// ---- POUs/_Grundfunktionen/FB_Heizregler.TcPOU
FUNCTION_BLOCK FB_Heizregler
VAR_INPUT
	diTempSoll	: DINT;
	diTempIst 	: DINT;
	iTimeOffs 	: INT; (* 0..99 *)
	iTimeGrp		: INT; (* Auswahl der Timer-Gruppe 0..9 *)
	iPMin 			: INT := 25;
	iPMax 			: INT := 100;
	iPHeizIn		: INT := 0;
	bNewData		: BOOL;
END_VAR
VAR_OUTPUT
	iPHeizOut : INT;
END_VAR
VAR
	bInitDone					 : BOOL;

	(* %I / %Q ********************)
	QbOutHeizSteller		AT %Q* : BOOL;
	bOutHeizSteller		: BOOL;

	dwPWMfast					: DWORD;

	iPWMTimer					: INT;
	iPHeiz						: INT;

	adiTempIst 				: ARRAY[0..2] OF DINT;
	diTempIstAend 		: DINT;

	diTempSollOld 		: DINT;
	diTempSollAend 		: DINT;

	diTempDiff 				: DINT;

	diResult_P				: DINT;
	diResult_I				: DINT;
	diResult_Dist			: DINT;
	diResult_Dsoll		: DINT;
	diResult					: DINT;
END_VAR

VAR PERSISTENT
	bManuell	: BOOL;
	iManPHeiz : INT;

	dikP			: DINT := 300; (* P-Regler, 1000 = 1.000 *)
	dikI			: DINT := 50; (* I-Regler, 1000 = 1.000 *)
	dikDist		: DINT := 5; (* D-Regler auf Istwert *)
	dikDsoll	: DINT := 5; (* D-Regler auf Sollwert => wirkt direkt auf I-Anteil *)

END_VAR

IF NOT bInitDone THEN
	M_Init();
END_IF

M_Ctrl();
M_PWM();
M_PWMfast();

ACTION M_Ctrl:
IF bNewData THEN
	diTempSollAend :=
			diTempSoll
		- diTempSollOld;
	diTempSollOld := diTempSoll;
	diTempIstAend :=
			diTempIst
		- adiTempIst[2];
	adiTempIst[2] := adiTempIst[1];
	adiTempIst[1] := adiTempIst[0];
	adiTempIst[0] := diTempIst;
END_IF

IF NOT bManuell
AND NOT (iPHeizIn > 0)
AND gbHeizGruppe[iTimeGrp]
THEN
	IF bNewData THEN
		diResult_Dist :=
				diTempIstAend
			* dikDist;

		diResult_Dsoll :=
				diTempSollAend
			* dikDsoll;

		diTempDiff :=
				diTempSoll
			- diTempIst
			+ diResult_Dist;

		diResult_P :=
				diTempDiff
			* dikP;

		diResult_I :=
				diTempDiff
			* dikI
			+ diResult_Dsoll
			+ diResult_I;
		IF (diResult_I
				> (100000 - diResult_P))
		THEN
			diResult_I :=
				(100000 - diResult_P);
		ELSIF (diResult_I < 0) THEN
			diResult_I := 0;
		END_IF

		diResult :=
				diResult_P
			+ diResult_I;
		iPHeiz := DINT_TO_INT(diResult / 1000);

	END_IF

ELSE
	diResult_I := iManPHeiz * 1000;
	iPHeiz := iManPHeiz;
END_IF
END_ACTION

ACTION M_PWMfast:
(* PWM im SPS-Zyklus *)
IF bOutHeizSteller THEN
	dwPWMfast := dwPWMfast + 1;
	IF (dwPWMfast > gdwPWMfast_88) THEN
		QbOutHeizSteller := TRUE;
						(*	 dwPWMfast.1
						OR dwPWMfast.2
						OR dwPWMfast.3;*)
	ELSIF (dwPWMfast > gdwPWMfast_75) THEN
		QbOutHeizSteller :=
							 dwPWMfast.1
						OR dwPWMfast.2;
	ELSE
		QbOutHeizSteller :=
							dwPWMfast.1;
	END_IF
	dwPWMfast := dwPWMfast AND 16#00FFFFFF;
ELSE
	QbOutHeizSteller := FALSE;
	dwPWMfast := INT_TO_DWORD(iTimeOffs / 10);
END_IF
END_ACTION

ACTION M_PWM:
(* PWM-Funktion *)
IF gbPWMTakt THEN
	IF bManuell THEN
		iPHeiz := iManPHeiz;
	ELSIF (iPHeizIn > 0) THEN
		iPHeiz := iPHeizIn;
	END_IF
	IF iPHeiz > iPMax THEN
		iPHeiz := iPMax;
	END_IF
	IF (giPWMTimer = iTimeOffs) THEN
		iPWMTimer := 0;
		IF (iPHeiz > 0) AND gbHeizGruppe[iTimeGrp] THEN
			bOutHeizSteller := TRUE;
		END_IF
	END_IF
	IF bOutHeizSteller THEN
		IF (iPWMTimer > (iPHeiz + iPMin)) THEN
			bOutHeizSteller := FALSE;
		END_IF
		iPWMTimer := iPWMTimer + 1;
	ELSE
		iPWMTimer := 0;
	END_IF
END_IF
iPHeizOut := iPHeiz;
END_ACTION

ACTION M_Init:
IF bNewData THEN
	diTempSollOld := diTempSoll;
	adiTempIst[2] := diTempIst;
	adiTempIst[1] := diTempIst;
	adiTempIst[0] := diTempIst;
	diResult_I := iManPHeiz * 1000;
	bInitDone := TRUE;
END_IF
END_ACTION

END_FUNCTION_BLOCK

// ---- POUs/_Grundfunktionen/FB_Heizregler_FBHR.TcPOU
(* Heizregler fuer Fussbodenheizung ueber Schaltventil und 
	Ruecklauftemperaturueberwachung (Schwallbetrie)
*)
FUNCTION_BLOCK FB_Heizregler_FBHR
VAR_INPUT
	INbEnable				: BOOL;
	INrTempSoll			: REAL;
	INrTempIst 			: REAL;
	INrTempVorlauf	: REAL; (* Temperatur, Heizung Vorlauf *)
	INrTempFBHR			: REAL; (* Temperatur, Fussbodenheizung Ruecklauf*)

	iTimeGrp				: INT; (* Auswahl der Timer-Gruppe 0..9 *)
	iPMin 					: INT := 25;
	iPMax 					: INT := 100;
	iPHeizIn				: INT := 0;
END_VAR
VAR_OUTPUT
	iPHeizOut : INT;
END_VAR
VAR
	bInitDone					 : BOOL;

	(* %I / %Q ********************)
	QbOutHeizSteller		AT %Q* : BOOL;
	bOutHeizSteller		: BOOL;


	tonCtrlCycle			: TON := (PT:=T#5S);
	bCtrlCycle				: BOOL;
	rPHeiz						: REAL;

	arTempIst 				: ARRAY[0..2] OF REAL;
	rTempIstAend 			: REAL;

	rTempSollOld 			: REAL;
	rTempSollAend 		: REAL;

	rTempDiff 				: REAL;

	rResult_P					: REAL;
	rResult_I					: REAL;
	rResult_Dist			: REAL;
	rResult_Dsoll			: REAL;
	rResult						: REAL;
	
	iOutputState			: INT; (* Status der Ausgangssteuerung *)
	iOutputCycleTime	: INT; (* Zeit [s] seit dem letzten Heizvorgang *)
	rOutputCycleTime	: REAL; (* Zeit [%] seit dem letzten Heizvorgang *)
	tonTimeCycle						: TON := (PT:= T#1S); (* Zeittakt *)
	tofWasserHeizung				: TOF := (PT:= T#3S); (* Mindest-Einschaltzeit *)
	tonVorlaufTemp					: TON := (PT:= T#5M); (* maximale Wartezeit auf Vorlauftemperatur *)
	tonVorlaufTempStop			: TON := (PT:= T#15M); (* Wartezeit, wenn Vorlauftemperatur zu gering war *)
	tonMinWartezeit					: TON := (PT:= T#3M); (* Mindest-Wartezeit nach einem Heizyklus bis zum naechsten Start *)

	rRueckTempStart		: REAL; (* Ruecklauftemperatur beim Start des akt. Heizzyklusses *)

END_VAR

VAR PERSISTENT
	bManuell					: BOOL;
	iManPHeiz 				: INT;
	iMaxCycleTime			: INT := 3600; (* maximale Heizzykluszeit [s] bei Heizleistung 1% *)

	rkP								: REAL := 300; (* P-Regler, 1000 = 1.000 *)
	rkI								: REAL := 50; (* I-Regler, 1000 = 1.000 *)
	rkDist						: REAL := 5; (* D-Regler auf Istwert *)
	rkDsoll						: REAL := 5; (* D-Regler auf Sollwert => wirkt direkt auf I-Anteil *)

	rVorlTempDiffMin	: REAL := 5.0; (* Mindestdifferenz zwischen Vorlauf- und Raumtemperatur *)
	rRueckTempDiffMax	: REAL := 5.0; (* Maximaler Temperaturanstieg im Ruecklauf zum Schliessen des Heizventils *)

END_VAR

IF NOT bInitDone THEN
	A_Init();
END_IF

tonCtrlCycle(IN:= NOT bCtrlCycle);
bCtrlCycle := tonCtrlCycle.Q;

A_Ctrl();
A_Output();

(* END *******************************)

ACTION A_Init:
rTempSollOld := INrTempSoll;
arTempIst[2] := arTempIst[1];
arTempIst[1] := arTempIst[0];
arTempIst[0] := INrTempIst;
rResult_I := iManPHeiz * 1000;
bInitDone := TRUE;

(* END *******************************)
END_ACTION

ACTION A_Output:
(* Zeittakt für Heizzyklus *)
tonTimeCycle(IN:= TRUE);
IF tonTimeCycle.Q THEN
	tonTimeCycle(IN:= FALSE);
	IF (iOutputCycleTime > 0) THEN
		iOutputCycleTime := iOutputCycleTime - 1;
	END_IF
END_IF
rOutputCycleTime :=
	iOutputCycleTime * 100
	/ iMaxCycleTime;
	

CASE iOutputState OF
0:
	QbOutHeizSteller := FALSE; 
	IF (rOutputCycleTime 
			< rPHeiz)
	AND (rPHeiz > 1.0) 
	THEN
		tofWasserHeizung(IN:= FALSE);
		tonVorlaufTemp(IN:= FALSE);
		tonVorlaufTempStop(IN:= FALSE);
		tonMinWartezeit(IN:= FALSE);
		rRueckTempStart :=
				INrTempFBHR;
		iOutputState := iOutputState + 1;
	END_IF

1: (* Heizzyklus aktiv, Ventil offen *)
	QbOutHeizSteller := TRUE; 
	tofWasserHeizung(IN:= TRUE);
	tonVorlaufTemp(IN:= TRUE);
	IF (INrTempFBHR
			> (rRueckTempStart + rRueckTempDiffMax))
	THEN (* Ruecklauftemperatur steigt an => Ventil schliessen *)
		iOutputState := iOutputState + 1;
	ELSIF tonVorlaufTemp.Q THEN
		IF (INrTempVorlauf
				< (INrTempFBHR
					+ rVorlTempDiffMin))
		THEN (* Vorlauftemperatur zu gering *)
			iOutputState := 10;
		ELSE (* max. Vorlaufzeit erreicht *)
			iOutputState := iOutputState + 1;
		END_IF
	END_IF

2: (* Heizzyklus beendet, Ventil schliessen *)
	QbOutHeizSteller := FALSE; 
	tonMinWartezeit(IN:= TRUE);
	IF tonMinWartezeit.Q THEN
		iOutputState := iOutputState + 1;
	END_IF

10: (* Vorlauftemperatur war zu gering *)
	QbOutHeizSteller := FALSE; 
	tonVorlaufTempStop(IN:= TRUE);
	IF tonVorlaufTempStop.Q THEN
		iOutputState := iOutputState + 1;
	END_IF

ELSE
	iOutputCycleTime := 
			iMaxCycleTime;
	iOutputState := 0;

END_CASE


(* END *******************************)
END_ACTION

ACTION A_Ctrl:
IF bCtrlCycle THEN
	rTempSollAend :=
			INrTempSoll
		- rTempSollOld;
	rTempSollOld := INrTempSoll;
	rTempIstAend :=
			INrTempIst
		- arTempIst[2];
	arTempIst[2] := arTempIst[1];
	arTempIst[1] := arTempIst[0];
	arTempIst[0] := INrTempIst;
END_IF

IF bManuell THEN
	rResult_I := iManPHeiz * 1000;
	rPHeiz := iManPHeiz;
	
ELSIF INbEnable
AND NOT (iPHeizIn > 0)
AND gbHeizGruppe[iTimeGrp]
THEN
	IF bCtrlCycle THEN
		rResult_Dist :=
				rTempIstAend
			* rkDist;

		rResult_Dsoll :=
				rTempSollAend
			* rkDsoll;

		rTempDiff :=
				INrTempSoll
			- INrTempIst
			+ rResult_Dist;

		rResult_P :=
				rTempDiff
			* rkP;

		rResult_I :=
				rTempDiff
			* rkI
			+ rResult_Dsoll
			+ rResult_I;
		IF (rResult_I
				> (100000 - rResult_P))
		THEN
			rResult_I :=
				(100000 - rResult_P);
		ELSIF (rResult_I < 0) THEN
			rResult_I := 0;
		END_IF

		rResult :=
				rResult_P
			+ rResult_I;
		rPHeiz := rResult / 1000;

	END_IF
END_IF

(* END *******************************)
END_ACTION

END_FUNCTION_BLOCK

// ---- POUs/_Grundfunktionen/FB_Licht.TcPOU
FUNCTION_BLOCK FB_Licht
VAR_INPUT
	bEinKurz				: BOOL;
	bEinLang				: BOOL;
	bAus 						: BOOL;
	tKurz						: TIME := t#5m;
	tLang 					: TIME := t#60m;
END_VAR
VAR_OUTPUT
END_VAR
VAR_IN_OUT
	bGruppeAus : BOOL;
END_VAR
VAR
	bInit 			: BOOL := TRUE;
	bInVisu			: BOOL;
	bIn					: BOOL;

	bKlickEnable	: BOOL;
	bLangEnable		: BOOL;

	(* %I / %Q ********************)
	IbInTaster		AT %I* : BOOL;
	QbOutLicht		AT %Q* : BOOL;

	tofEin			: TOF;

	fbTaster 		: FB_Taster;

  fbLog : FB_LoggerSetMsg;
END_VAR

IF bInit THEN
	bKlickEnable := (tkurz <> t#0s);
	bLangEnable := (tLang <> t#0s);
	bInit := FALSE;
END_IF


bIn := IbInTaster OR bInVisu;
fbTaster(bIn:= bIn);

IF bKlickEnable
AND (fbTaster.bKlick
		OR bEinKurz
		OR gbLichtZentralEin)
THEN
	tofEin(IN:= TRUE, PT:= tkurz);
ELSIF bLangEnable
AND (fbTaster.bLang
		OR bEinLang)
THEN
	tofEin(IN:= TRUE, PT:= tLang);
END_IF
tofEin(IN:= FALSE);

IF fbTaster.bLang AND bKlickEnable AND bLangEnable THEN
  IF NOT QbOutLicht THEN
    fbLog.M_AddMsgHint('Licht EIN Taster');
  END_IF
	QbOutLicht := TRUE;
ELSIF bEinKurz OR bEinLang THEN
  IF NOT QbOutLicht THEN
    fbLog.M_AddMsgHint('Licht EIN INPUT');
  END_IF
	QbOutLicht := TRUE;
ELSIF gbLichtZentralEin THEN
	QbOutLicht := TRUE;
  //fbLog.M_AddMsgHint('Licht EIN ZentralEin');
END_IF

IF (fbTaster.bKlick
		AND bKlickEnable)
OR (fbTaster.bLang
		AND NOT bKlickEnable
		AND bLangEnable)
THEN
  IF NOT QbOutLicht THEN
    IF NOT QbOutLicht THEN
      fbLog.M_AddMsgHint('Licht EIN Taster');
    END_IF
  	QbOutLicht := TRUE;
  ELSE
    IF QbOutLicht THEN
      fbLog.M_AddMsgHint('Licht AUS Taster');
    END_IF
  	QbOutLicht := FALSE;
  END_IF
END_IF

IF QbOutLicht AND NOT tofEin.Q THEN
  IF QbOutLicht THEN
    fbLog.M_AddMsgWarning('Licht AUS Taster');
  END_IF
	QbOutLicht := FALSE;
ELSIF bAus THEN
  IF QbOutLicht THEN
    fbLog.M_AddMsgWarning('Licht AUS INPUT');
  END_IF
	QbOutLicht := FALSE;
ELSIF gbLichtZentralAus THEN
	QbOutLicht := FALSE;
  //fbLog.M_AddMsgHint('Licht AUS ZentralAus');
END_IF

IF fbTaster.bKlick2 THEN
	bGruppeAus := TRUE;
END_IF

END_FUNCTION_BLOCK

// ---- POUs/_Grundfunktionen/FB_Rollo.TcPOU
FUNCTION_BLOCK FB_Rollo
VAR_INPUT
	bInTasterAuf 			: BOOL;
	bInTasterAb				: BOOL;
	bCfgTimeAb				: BOOL; (* Rollo ab, bei globaler Schaltzeit *)
	bCfgTimeAbWinter	: BOOL; (* Rollo ab, bei globaler Schaltzeit, aber nur waehrend Winderzeit *)
	itGesamt					: INT; (* x 100ms *)
	itSchatten				: INT; (* x 100ms *)
END_VAR
VAR_OUTPUT
	bOutRollo			: BOOL;
END_VAR
VAR_IN_OUT
	bAbVorw	: BOOL;
	bAb			: BOOL;
END_VAR
VAR
	bInVisuAuf 	: BOOL;
	bInVisuAb		: BOOL;
	bOutVisuAb	: BOOL;
	bInAuf 			: BOOL;
	bInAb				: BOOL;

	iRolloMode 	: E_RolloMode;
	bTaster			: BOOL;
	bTasterAb		: BOOL;
	bRollo			: BOOL;
	bAbVorwi	: BOOL;
	iActPos			: INT;

	tofLock		: TOF := (PT:= t#50ms);
	fbTaster	: FB_Taster;


	tonSwitch		: TON := (PT:= t#100ms);
	tonStart		: TON := (PT:= t#50ms);


END_VAR

bInAuf := bInTasterAuf
				OR bInVisuAuf
				OR (bCfgTimeAb
						AND gbTimeRolloAuf);
bInAb := bInTasterAb
				OR bInVisuAb
				OR (bCfgTimeAb
						AND gbTimeRolloAb
						AND (NOT bCfgTimeAbWinter
								OR NOT gfbSystemCX.OUTbSummerTime));
bOutVisuAb := bAb;

IF bInAuf AND bInAb THEN
	tofLock.IN := TRUE;
ELSIF NOT bInAuf AND NOT bInAb THEN
	tofLock.IN := FALSE;
END_IF
tofLock();

bTaster := (bInAuf XOR bInAb) AND NOT tofLock.Q;
IF bTaster THEN
	bTasterAb := bInAb;
END_IF
fbTaster(bIn:= bTaster);


IF NOT tofLock.Q THEN
	IF fbTaster.bLang THEN
		iRolloMode := eRollo_Manuell;
	ELSIF fbTaster.bKlick THEN
		IF iRolloMode > eRollo_Stop THEN
			iRolloMode := eRollo_Stop;
		ELSE
			iRolloMode := eRollo_Auto;
		END_IF
	ELSIF fbTaster.bKlick2 THEN
		iRolloMode := eRollo_Schatten;
	END_IF
END_IF

CASE iRolloMode OF
eRollo_Stop:
	IF (iActPos < 0) THEN
		iActPos := 0;
	END_IF

eRollo_Manuell:
	IF NOT bTaster THEN
		iRolloMode := eRollo_Stop;
	END_IF

eRollo_Auto:
	IF bRollo AND NOT bTaster THEN
		IF bAbVorwi THEN
			IF (iActPos > itGesamt) THEN
				iRolloMode := eRollo_Stop;
			END_IF
		ELSE
			IF (iActPos < -30) THEN
				iRolloMode := eRollo_Stop;
			END_IF
		END_IF
	END_IF

eRollo_Schatten:
	IF bRollo THEN
		IF NOT bAbVorwi THEN
			IF (iActPos < itSchatten) THEN
				iRolloMode := eRollo_Stop;
			END_IF
		ELSE
			IF (iActPos > itSchatten) THEN
				iRolloMode := eRollo_Stop;
			END_IF
		END_IF
	END_IF

END_CASE

IF (iActPos > itGesamt) THEN
	iActPos := itGesamt;
ELSIF (iActPos < -30) THEN
	iActPos := -30;
END_IF


IF NOT bRollo AND (iRolloMode > eRollo_Stop) THEN
	bRollo := TRUE;
	bAbVorw := bTasterAb;
	bAbVorwi := bAbVorw;
ELSIF (bOutRollo AND (bAbVorwi <> bAb)) THEN
	tofLock.IN := TRUE;
	iRolloMode := eRollo_Stop;
	bRollo := FALSE;
ELSIF (bRollo AND (iRolloMode = eRollo_Stop)) THEN
	tofLock.IN := TRUE;
	iRolloMode := eRollo_Stop;
	bRollo := FALSE;
END_IF

tonSwitch(IN:= bRollo);
tonStart(IN:= tonSwitch.Q);

IF tonSwitch.Q THEN
	bAb := bAbVorw;
END_IF
bOutRollo := tonStart.Q;

IF bOutRollo AND gbTakt100ms THEN
	IF bAb THEN
		iActPos := iActPos + 1;
	ELSE
		iActPos := iActPos - 1;
	END_IF
END_IF

END_FUNCTION_BLOCK

// ---- POUs/_Grundfunktionen/FB_RolloGruppe.TcPOU
FUNCTION_BLOCK FB_RolloGruppe
VAR_INPUT
	bCfgTimeAb				: BOOL; (* Rollo ab, bei globaler Schaltzeit *)
	bCfgTimeAbWinter	: BOOL; (* Rollo ab, bei globaler Schaltzeit, aber nur waehrend Winderzeit *)
	iAnzRollo					: INT := 1;
	aitGesamt 				: ARRAY[1..3] OF INT;
	aitSchatten 			: ARRAY[1..3] OF INT;
END_VAR
VAR_OUTPUT

END_VAR
VAR
	bInit 			: BOOL := TRUE;
	bInVisuAuf 	: BOOL;
	bInVisuAb		: BOOL;
	bInAuf 			: BOOL;
	bInAb				: BOOL;

	iArr				: INT;

	(* %I / %Q ********************)
	IbInTasterAuf		AT %I* : BOOL;
	IbInTasterAb	 	AT %I* : BOOL;
	QbOutRolloAb		AT %Q* : BOOL;
	QbOutRollo1	 		AT %Q* : BOOL;
	QbOutRollo2	 		AT %Q* : BOOL;
	QbOutRollo3	 		AT %Q* : BOOL;

	(* Rollosteuerung *)
	bAbVorw 		: BOOL;
	bAb					: BOOL;

	fbRollo 		: ARRAY[1..3] OF FB_Rollo;
	tonRolloAb	: TON := (PT:= t#30s);

  fbLog : FB_LoggerSetMsg;
	bLogMsgAuf : BOOL;
	bLogMsgAb : BOOL;
END_VAR

IF bInit THEN
	bInit := FALSE;
	FOR iArr := 1 TO 3 DO
		fbRollo[iArr].bCfgTimeAb := bCfgTimeAb;
		IF (iArr = 3) THEN (* soll nur fuer 3. Rollo im Esszimmer gelten = Tuere *)
			fbRollo[iArr].bCfgTimeAbWinter := bCfgTimeAbWinter;
		END_IF
		fbRollo[iArr].itGesamt := aitGesamt[iArr];
		fbRollo[iArr].itSchatten := aitSchatten[iArr];
	END_FOR
END_IF

bInAuf := IbInTasterAuf OR bInVisuAuf;
bInAb := IbInTasterAb OR bInVisuAb;

fbRollo[1](
	bInTasterAuf:= bInAuf,
	bInTasterAb:= bInAb,
	bAbVorw:= bAbVorw,
	bAb:= bAb,
	bOutRollo=> QbOutRollo1);

IF iAnzRollo >=2 THEN
	fbRollo[2](
		bInTasterAuf:= bInAuf,
		bInTasterAb:= bInAb,
		bAbVorw:= bAbVorw,
		bAb:= bAb,
		bOutRollo=> QbOutRollo2);
END_IF

IF iAnzRollo >=3 THEN
	fbRollo[3](
		bInTasterAuf:= bInAuf,
		bInTasterAb:= bInAb,
		bAbVorw:= bAbVorw,
		bAb:= bAb,
		bOutRollo=> QbOutRollo3);
END_IF

QbOutRolloAb := bAb;

tonRolloAb(IN:= QbOutRolloAb AND NOT (QbOutRollo1 OR QbOutRollo2 OR QbOutRollo3));
IF tonRolloAb.Q THEN
	bAbVorw := FALSE;
	bAb := FALSE;
END_IF

// Log Meldungen
IF NOT bLogMsgAuf AND bInAuf AND NOT QbOutRolloAb
AND (QbOutRollo1 OR QbOutRollo2 OR QbOutRollo3)
THEN
  fbLog.M_AddMsgHint('Rollo AUF Taster');
  bLogMsgAuf := TRUE;
ELSE
  bLogMsgAuf := FALSE;
END_IF
IF NOT bLogMsgAb AND bInAb AND QbOutRolloAb
AND (QbOutRollo1 OR QbOutRollo2 OR QbOutRollo3)
THEN
  fbLog.M_AddMsgHint('Rollo AB Taster');
  bLogMsgAb := TRUE;
ELSE
  bLogMsgAb := FALSE;
END_IF

END_FUNCTION_BLOCK

// ---- POUs/_Grundfunktionen/FB_TasterProg.TcPOU
FUNCTION_BLOCK FB_TasterProg
VAR_INPUT
	bCfgRollo 	: BOOL;
	bIn 		: BOOL;
END_VAR

VAR_OUTPUT
	bKlick			: BOOL;
	bKlick2			: BOOL;
	bKlick3			: BOOL;
	bLang				: BOOL;
	bProg				: BOOL;
	iKlick			: INT;
	iProgCode		: INT;
END_VAR
VAR
	bKlick_i		: BOOL;

	iProgState	: INT;
	iKlickCnt		: INT;
	iCode1			: INT;
	iCode10			: INT;

	tofPrell 		: TOF := (PT:= t#30ms);
	tofKlick 		: TOF := (PT:= t#200ms);
	tonLang 		: TON := (PT:= t#500ms);
	tonProg 		: TON := (PT:= t#3s);
	tofProg	 		: TOF := (PT:= t#5s);

	rtrigTast	 	: R_TRIG;
	ftrigKlick 	: F_TRIG;
	rtrigLang  	: R_TRIG;

END_VAR

tofPrell(IN:= bIn);
rtrigTast(CLK:= tofPrell.Q);
bKlick_i := rtrigTast.Q AND NOT tofKlick.Q;

tofKlick(IN:= rtrigTast.Q);
ftrigKlick(CLK:= tofKLick.Q);

IF rtrigTast.Q THEN
	iKlickCnt := iKlickCnt + 1;
END_IF

CASE iProgState OF
0: (* normal: *)
	tonLang(IN:= tofPrell.Q);
	rtrigLang(CLK:= tonLang.Q);

	tonProg(IN:= tofPrell.Q);
	IF tonProg.Q THEN
		tofProg(IN:= FALSE);
		tofProg(IN:= TRUE);
		iProgState := iProgState + 1;
		iKlickCnt := 0;
	END_IF

1: (* Progstatus, Codewert x10 *)
	IF ftrigKlick.Q THEN
		IF iKlickCnt = 0 THEN
			iProgState := 0;
		ELSE
			iCode10 := iKlickCnt;
			iKlickCnt := 0;
			iProgState := iProgState + 1;
		END_IF
	END_IF

2: (* Progstatus, Codewert x1 *)
	IF ftrigKlick.Q THEN
		IF iKlickCnt = 0 THEN
			iProgState := 0;
		ELSE
			iCode1 := iKlickCnt;
			iKlickCnt := 0;
			iProgState := iProgState + 1;
		END_IF
	END_IF

3: (* Codewertausgabe *)
	iProgCode := iCode10 * 10 + iCode1;
	iProgState := iProgState + 1;

4:
	iProgCode := 0;
	iProgState := 0;

END_CASE


(* Ausgabe *)
CASE iProgState OF
0:
	bProg := FALSE;
	iProgCode	:= 0;

	bKlick := bKlick_i;
	IF ftrigKlick.Q THEN
		iKlick := iKlickCnt;
		bKlick2 := iKlick = 2;
		bKlick3 := iKlick = 3;
		iKlickCnt := 0;
	ELSE
		iKlick := 0;
		bKlick2 := FALSE;
		bKlick3 := FALSE;
	END_IF

	IF bCfgRollo THEN
		bLang := tonLang.Q;
	ELSE
		bLang := rtrigLang.Q;
	END_IF


ELSE
	bKlick := FALSE;
	bKlick2 := FALSE;
	bKlick3 := FALSE;
	bLang := FALSE;
	bProg := TRUE;
	iKlick := 0;

	tofProg(IN:= rtrigTast.Q);
	IF NOT tofProg.Q THEN
		iProgState := 0;
	END_IF

END_CASE

END_FUNCTION_BLOCK

// ---- POUs/_Grundfunktionen/F_Scaling.TcPOU
FUNCTION F_Scaling : DINT
VAR_INPUT
	diInput 	: DINT;
	diRef100 	: DINT;
END_VAR


VAR
END_VAR
(*All VAR_IN_OUT variables have been moved to the end of the declaration due to compatibility reasons*)
VAR_IN_OUT
	stScal 		: ST_AnalogScaling;
END_VAR

F_Scaling :=
		(diInput
		- stScal.diXRef)
	* stScal.diFact
	/ diRef100
	+ stScal.diYRef;

END_FUNCTION

// ---- GlobalTextList.TcGTLO
TEXTLIST GlobalTextList
  181 = '\n\n'
  175 = '\nKompressorsteuerung'
  162 = '\n\n\nLufttrockner'
  165 = '\nKompressor'
  163 = '\nLufttrockner'
  164 = '\nNotkompressor'
  197 = ' \t\t\t1: Puffer4000_unten\n\t\t\t2: Puffer4000_mitte\n\t\t\t3: Puffer4000_oben\n\t\t\t4: Puffer4000_Brauchw *)\n '
  242 = '   Filter black list:'
  247 = '   Filter white list:'
  237 = '   Meldungen:'
  35 = '  %s'
  200 = '  1: Puffer4000_unten\n  2: Puffer4000_mitte\n  3: Puffer4000_oben\n  4: Puffer4000_Brauchw'
  18 = '  Ankleide'
  218 = '  Ausschaltverzögerung kurz:'
  17 = '  Bad'
  27 = '  Büro'
  21 = '  Diele'
  26 = '  Essen'
  31 = '  Heizung'
  32 = '  Hobby'
  20 = '  Kind1'
  16 = '  Kind2'
  15 = '  Kind3'
  25 = '  Kochen'
  105 = '  Raum'
  30 = '  Sauna'
  19 = '  Schlafen'
  22 = '  Speiss'
  34 = '  Vorrat'
  33 = '  Waschen'
  106 = '  Wasser'
  14 = '  WC'
  28 = '  Wohnen'
  190 = ' $IN_Title$:'
  220 = ' %d'
  0 = ' %s'
  193 = ' %s:'
  43 = ' - AUS: '
  44 = ' - EIN: '
  37 = ' - Rollo AB:'
  38 = ' - Rollo AUF:'
  199 = ' 1: Puffer4000_unten\n 2: Puffer4000_mitte\n 3: Puffer4000_oben\n 4: Puffer4000_Brauchw'
  198 = ' 1: Puffer4000_unten\n 2: Puffer4000_mitte\n 3: Puffer4000_oben\n 4: Puffer4000_Brauchw\n '
  279 = ' Auswahl des Temperatursensors \n zur Steuerung der Pufferumwaelzpumpe \n zum Wohnhaus/Werkstatt :'
  201 = ' Auswahl des Temperatursensors \n zur Steuerung der Pufferumwaelzpumpe \n zum Wohnhaus/Werkstatt :'
  196 = ' Auswahl des Temperatursensors \n zur Steuerung der Pufferumwaelzpumpen \n zum Wohnhaus/Werkstatt '
  283 = ' Auswahl des Temperatursensors zur Steuerung der \nPufferumwaelzpumpe zum Wohnhaus/Werkstatt'
  281 = ' Auswahl des Temperatursensors zur Steuerung der \nPufferumwaelzpumpe zum Wohnhaus/Werkstatt :'
  280 = ' Auswahl des Temperatursensors zur Steuerung der Pufferumwaelzpumpe zum Wohnhaus/Werkstatt :'
  258 = ' Auswertung gestartet ab Logeintrag: %s'
  53 = ' Büro'
  52 = ' Essen, Kochen, Diele\n EG/OG, WCs, Hobby,\n Sauna'
  259 = ' Filter:'
  191 = ' IN_Title:'
  278 = ' Kellerräume:'
  189 = ' KG WC-Herren:'
  186 = ' KG WC-Räume:'
  50 = ' Kinderzimmer'
  270 = ' Letzter Logeintrag in Datei: %s'
  257 = ' Letzter Logeintrag: %s'
  265 = ' Log-Datei: %s_ n.csv'
  57 = ' Manuell'
  256 = ' Message (Datum, Uhrzeit, Pfad, Text)'
  187 = ' Nachlaufzeit Abluftventilator'
  271 = ' Nicht gespeicherte Logeinträge: %s'
  104 = ' Raum'
  45 = ' Schaltzeiten Heizgruppe 0:'
  46 = ' Schaltzeiten Heizgruppe 1:'
  47 = ' Schaltzeiten Heizgruppe 2:'
  48 = ' Schaltzeiten Heizgruppe 3:'
  49 = ' Schaltzeiten Heizgruppe 4:'
  39 = ' Schaltzeiten Rollos:'
  54 = ' Schlafzimmer'
  42 = ' Uhrzeit stellen:'
  51 = ' Wohnzimmer, Bad OG,\n Bad EG (Heizkörper)\n Sauna (Heizkörper)'
  141 = '%1.2f'
  140 = '%1.2f%%'
  145 = '%1.3f'
  117 = '%2.1f'
  114 = '%2.1f%'
  58 = '%2.1f°C'
  157 = '%3.1f %'
  179 = '%3.1f C'
  152 = '%3.1f °C'
  178 = '%3.1f°C'
  143 = '%3.2f'
  62 = '%i'
  60 = '%s'
  241 = '%s '
  219 = '%s min'
  188 = '%s sek'
  56 = '%s%%'
  263 = '&'
  252 = "'black list: Begriff1[;Begriff2[;Begriff3]]'"
  248 = "'whitelist: Begriff1[;Begriff2[;Begriff3]]'"
  123 = '+'
  124 = '-'
  253 = '...'
  262 = '/'
  89 = '1'
  202 = '1: '
  284 = '2'
  204 = '2: '
  285 = '3'
  205 = '3: '
  286 = '4'
  206 = '4: '
  287 = '5'
  207 = '5: '
  288 = '6'
  208 = '6: '
  289 = '7'
  290 = '8'
  112 = '<'
  113 = '<<'
  111 = '>'
  110 = '>>'
  120 = '>]'
  118 = '>|'
  8 = 'AB'
  41 = 'Aktuelle Uhrzeit kopieren'
  95 = 'Alarm'
  296 = 'ALARM'
  306 = 'Alarm quittieren'
  307 = 'Alarm quittieren\nund Transoren\nstarten'
  249 = 'Alle'
  7 = 'AUF'
  2 = 'AUS'
  217 = 'Ausschaltverzögerung kurz:'
  216 = 'Ausschaltverzögerung lang:'
  195 = 'Auswahl des Temperatursensors \nzur Steuerung der Pufferumwaelzpumpen \nzum Wohnhaus/Werkstatt '
  194 = 'Auswahl des Temperatursensors zur Steuerung der Pufferumwaelzpumpen zum Wohnhaus/Werkstatt '
  138 = 'Auto'
  149 = 'Auto revers'
  135 = 'Beckenstrahler'
  9 = 'Beenden'
  148 = 'Beleuchtung'
  136 = 'Betriebsart RGB'
  212 = 'Bewegungsmelder-Licht: Schaltzeiten fuer lange Ausschaltverzögerung '
  211 = 'bis'
  214 = 'bis Wochentag'
  264 = 'black'
  11 = 'Dachgeschoss'
  273 = 'Das Klemmen-Bus-System\nwird neu gestartet!\n\nEs werden für wenige Sekunden\n alle Ausgänge abgeschaltet\n(z.B. Lichter...).'
  269 = 'Daten sofort speichern'
  268 = 'Daten speichern'
  267 = 'Daten werden automatisch gespeichert,\nwenn eine Mindestanzahl ungespeicherter\nMeldungen vorhanden ist.'
  266 = 'Datenspeicherung aktivieren'
  130 = 'Decke Nord RGB'
  131 = 'Decke Nord W'
  132 = 'Decke Nord WEISS'
  125 = 'Decke Süd'
  126 = 'Decke Süd\nRGB'
  127 = 'Decke Süd \nRGB'
  128 = 'Decke Süd RGB'
  129 = 'Decke Süd W'
  133 = 'Decke Süd WEISS'
  244 = 'del'
  78 = 'DG'
  222 = 'Di'
  230 = 'Dienstag'
  61 = 'DMX 512 Light Control'
  224 = 'Do'
  232 = 'Donnerstag'
  96 = 'Druckt.'
  79 = 'EG'
  55 = 'EIN'
  3 = 'EIN '
  94 = 'Ein/Aus'
  10 = 'Einstellungen'
  12 = 'Erdgeschoss'
  260 = 'Error'
  274 = 'Es wird ein Neustart\nder Steuerung durchgeführt!\n\nDie Steuerung wird während\ndes Neustarts für ca. 1 Minute\nnicht erreichbar sein.'
  142 = 'Farbe'
  65 = 'FAST'
  99 = 'FBHeiz.Rückl.'
  88 = 'FBHeiz.Rücklauf'
  251 = 'Fehlermeldungen'
  90 = 'Filterpumpe'
  203 = 'Filterpumpe, Schaltzeiten'
  225 = 'Fr'
  233 = 'Freitag'
  92 = 'Gegenstromanl.'
  144 = 'Geschwindigkeit'
  71 = 'Hauptseite (PC)'
  87 = 'Heizung Vorlauf'
  139 = 'Helligkeit'
  97 = 'Hy'
  116 = 'Hygro'
  255 = 'Id'
  192 = 'IN_Title'
  82 = 'Ist'
  13 = 'Keller'
  282 = 'Kellerräume'
  277 = 'Kellerräume:'
  77 = 'KG'
  185 = 'KG WC-Räume:'
  310 = 'Klemmen-\nBus-System \nneu starten'
  309 = 'Klemmen-Bus-System \nneu starten'
  236 = 'Klemmen-Bus-System neu starten'
  93 = 'Klimagerät'
  158 = 'Kompressor'
  176 = 'Kompressorsteuerung'
  59 = 'L'
  4 = 'Licht'
  1 = 'Licht DG'
  5 = 'Licht KG'
  297 = 'Liquiphanten'
  291 = 'Liquiphanten Konfiguration'
  160 = 'Lufttrockner'
  161 = 'Lufttrockner\n'
  245 = 'löschen'
  72 = 'Main'
  137 = 'Manuell'
  223 = 'Mi'
  231 = 'Mittwoch'
  221 = 'Mo'
  73 = 'Mobile'
  275 = 'Monitoring'
  229 = 'Montag'
  184 = 'Nach Abschalten des Bewegungsmelders \nläuft der Abluftventilator die hier \neingestellte Zeit nach'
  183 = 'Nachlaufzeit Abluftventilator'
  294 = 'Name'
  36 = 'Neue Uhrzeit setzen'
  298 = 'Not-Aus'
  159 = 'Notkompressor'
  292 = 'Nr'
  295 = 'Nr %s'
  122 = 'OK'
  74 = 'PC'
  151 = 'Puffer\n4000l'
  174 = 'Puffer\n4000l\n\n'
  153 = 'Puffer\n4000l\n\n\n\n'
  154 = 'Puffer\n4000l\n\n\n\n\n\n'
  173 = 'Puffer\nWerkstatt\n\n\n'
  182 = 'Puffer\nWerkstatt\n\n\n\n\n'
  156 = 'Puffer\nWerkstatt\n\n\n\n\n\n'
  172 = 'Puffer\nWohnhaus\n\n\n'
  180 = 'Puffer\nWohnhaus\n\n\n\n\n'
  155 = 'Puffer\nWohnhaus\n\n\n\n\n\n'
  86 = 'Raum'
  84 = 'Raum:'
  6 = 'Rollo'
  69 = 'Rot'
  303 = 'Rückmeldekont.1'
  304 = 'Rückmeldekont.2'
  226 = 'Sa'
  234 = 'Samstag'
  80 = 'ScB'
  209 = 'Schaltzeiten Beleuchtung Bewegunsmelder'
  215 = 'Schaltzeiten fuer lange Ausschaltverzögerung '
  302 = 'Schlüsselschalter'
  102 = 'Schw-\nbad'
  107 = 'Schwi-\nbad'
  101 = 'Schwimm-\nbad'
  67 = 'Schwimmbad'
  146 = 'Schwimmbad Beleuchtung'
  76 = 'Schwimmbad Licht'
  68 = 'Schwimmbad RGBW'
  109 = 'Schwimmbad Soll-Temperatur'
  300 = 'Sensor'
  66 = 'SLOW'
  227 = 'So'
  81 = 'Soll'
  103 = 'Soll-Temperatur'
  168 = 'Solltemperatur\nVorlauf'
  40 = 'Sommerzeit'
  228 = 'Sonntag'
  70 = 'Speed'
  64 = 'Speed: %i'
  272 = 'Speichern auf Netzwerkpfad'
  254 = 'speichern/laden'
  177 = 'Start'
  301 = 'Start/\nQuit'
  63 = 'Start/Stop'
  108 = 'Startseite'
  308 = 'Steuerung \nneu starten'
  235 = 'Steuerung neu starten'
  91 = 'Strömungswächter'
  171 = 'Störung'
  75 = 'szUeberschrift'
  239 = 'TcRestart:'
  115 = 'Temp'
  83 = 'Temperatur'
  166 = 'Temperatur, Umschaltung'
  167 = 'Temperatur, Umschaltung\nSchnellaufladung'
  169 = 'Temperatur, Umschaltung\nzum Wohnhaus'
  170 = 'Temperatur, Umschaltung\nzur Werkstatt'
  98 = 'Tmp'
  23 = 'Tor 1\noffen'
  24 = 'Tor 2\noffen'
  305 = 'Transor Start'
  293 = 'Transorauswahl'
  299 = 'Transoren'
  100 = 'V'
  29 = 'VISU wurde beendet.'
  210 = 'von'
  213 = 'von Wochentag'
  134 = 'Wandleuchten'
  250 = 'Warnungen'
  85 = 'Wasser'
  147 = 'WEISS\n%i'
  261 = 'white'
  243 = 'whitelist: Begriff1[;Begriff2[;Begriff3]]'
  238 = 'X'
  121 = 'ZURÜCK'
  246 = 'zurück'
  240 = 'Zähler:'
  119 = '[<'
  150 = 'Übersicht'
  276 = 'Überwachungen'
END_TEXTLIST

// ---- Logger/VISUs/V_LoggerFilterBlack.TcVIS
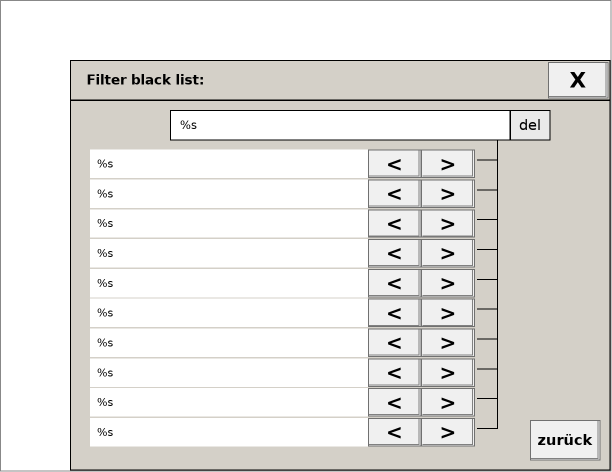
VISUALIZATION V_LoggerFilterBlack  // 612x472
    Rectangle (70,100 540x370)
    Rectangle (70,60 540x40), "Filter black list:"
    Frame (80,130 420x320)
        shows V_LoggerFilterList(IOfbLogger := gfbLogger, IOszFilterTxt := gfbLogger.szVisuFilterBlack)
    Rectangle (170,110 340x30), "%s", tooltip "whitelist: Begriff1[;Begriff2[;Begriff3]]", text variable: gfbLogger.szVisuFilterBlack
        OnMouseClick: write the text variable via Default
    Rectangle (510,110 40x30), "del", tooltip "löschen"
        OnMouseClick: execute { gfbLogger.szVisuFilterBlack := ''; }
    Button (530,420 70x40), "zurück"
        OnMouseClick: change screen: Previous 
    Button (548,62 60x36), "X"
        OnMouseClick: change screen: Previous 
END_VISUALIZATION

// ---- Logger/VISUs/V_LoggerFilterLine.TcVIS
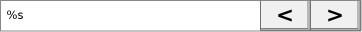
VISUALIZATION V_LoggerFilterLine  // 362x32
VAR_IN_OUT
	IOszTxtActual : STRING(80);
	IOszTxtLine : STRING(80);
END_VAR
    Rectangle (0,0 260x30), "%s", text variable: IOszTxtLine
        OnMouseClick: write the text variable via Default
    Button (260,0 50x30), "<"
        OnMouseClick: execute { IOszTxtLine := IOszTxtActual; }
    Button (310,0 50x30), ">"
        OnMouseClick: execute { IOszTxtActual := IOszTxtLine; }
END_VISUALIZATION

// ---- Logger/VISUs/V_LoggerFilterList.TcVIS
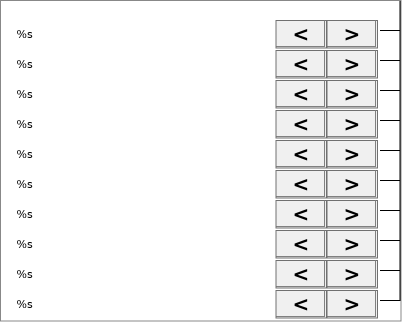
VISUALIZATION V_LoggerFilterList  // 402x322
VAR_IN_OUT
  IOfbLogger : FB_Logger;
	IOszFilterTxt : STRING(80);
END_VAR
    Line (400,300) (400,0)
    Frame (10,20 370x30)
        shows V_LoggerFilterLine(IOszTxtActual := IOszFilterTxt, IOszTxtLine := IOfbLogger.anvszVisuFilter[1])
    Frame (10,50 370x30)
        shows V_LoggerFilterLine(IOszTxtActual := IOszFilterTxt, IOszTxtLine := IOfbLogger.anvszVisuFilter[2])
    Frame (10,80 370x30)
        shows V_LoggerFilterLine(IOszTxtActual := IOszFilterTxt, IOszTxtLine := IOfbLogger.anvszVisuFilter[3])
    Frame (10,110 370x30)
        shows V_LoggerFilterLine(IOszTxtActual := IOszFilterTxt, IOszTxtLine := IOfbLogger.anvszVisuFilter[4])
    Frame (10,140 370x30)
        shows V_LoggerFilterLine(IOszTxtActual := IOszFilterTxt, IOszTxtLine := IOfbLogger.anvszVisuFilter[5])
    Line (380,30) (400,30)
    Line (380,60) (400,60)
    Line (380,90) (400,90)
    Line (380,120) (400,120)
    Line (380,150) (400,150)
    Frame (10,170 370x30)
        shows V_LoggerFilterLine(IOszTxtActual := IOszFilterTxt, IOszTxtLine := IOfbLogger.anvszVisuFilter[6])
    Frame (10,200 370x30)
        shows V_LoggerFilterLine(IOszTxtActual := IOszFilterTxt, IOszTxtLine := IOfbLogger.anvszVisuFilter[7])
    Frame (10,230 370x30)
        shows V_LoggerFilterLine(IOszTxtActual := IOszFilterTxt, IOszTxtLine := IOfbLogger.anvszVisuFilter[8])
    Frame (10,260 370x30)
        shows V_LoggerFilterLine(IOszTxtActual := IOszFilterTxt, IOszTxtLine := IOfbLogger.anvszVisuFilter[9])
    Frame (10,290 370x30)
        shows V_LoggerFilterLine(IOszTxtActual := IOszFilterTxt, IOszTxtLine := IOfbLogger.anvszVisuFilter[10])
    Line (380,180) (400,180)
    Line (380,210) (400,210)
    Line (380,240) (400,240)
    Line (380,270) (400,270)
    Line (380,300) (400,300)
END_VISUALIZATION

// ---- Logger/VISUs/V_LoggerFilterWhite.TcVIS
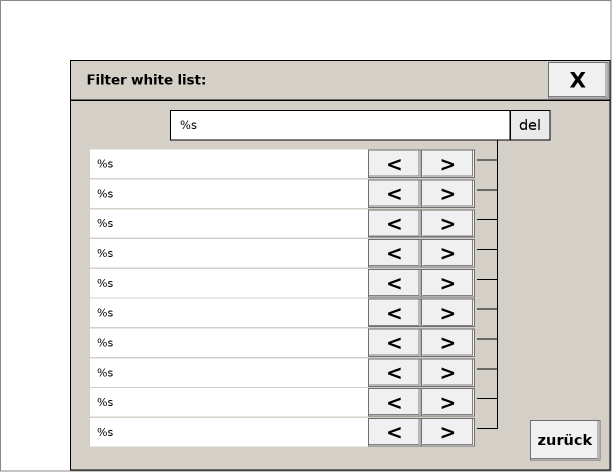
VISUALIZATION V_LoggerFilterWhite  // 612x472
    Rectangle (70,100 540x370)
    Rectangle (70,60 540x40), "Filter white list:"
    Frame (80,130 420x320)
        shows V_LoggerFilterList(IOfbLogger := gfbLogger, IOszFilterTxt := gfbLogger.szVisuFilterWhite)
    Rectangle (170,110 340x30), "%s", tooltip "whitelist: Begriff1[;Begriff2[;Begriff3]]", text variable: gfbLogger.szVisuFilterWhite
        OnMouseClick: write the text variable via Default
    Rectangle (510,110 40x30), "del", tooltip "löschen"
        OnMouseClick: execute { gfbLogger.szVisuFilterWhite := ''; }
    Button (530,420 70x40), "zurück"
        OnMouseClick: change screen: Previous 
    Button (548,62 60x36), "X"
        OnMouseClick: change screen: Previous 
END_VISUALIZATION

// ---- Logger/VISUs/V_LoggerModul.TcVIS
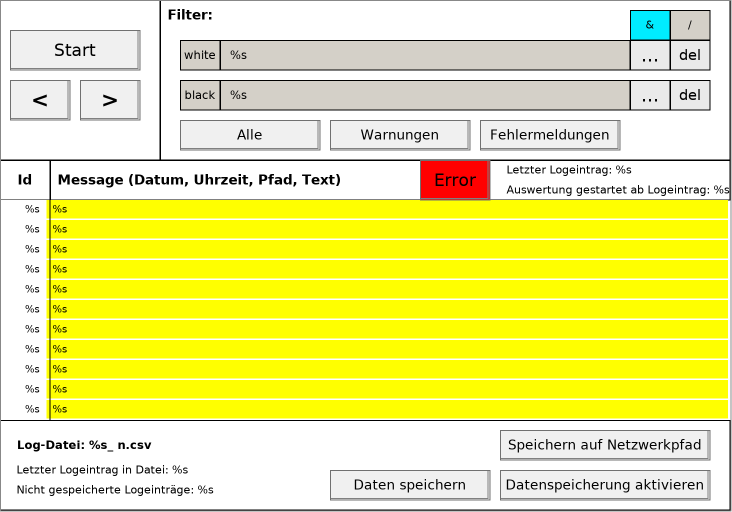
VISUALIZATION V_LoggerModul  // 732x512
VAR_IN_OUT
  fbLogger : FB_Logger;
END_VAR
    Rectangle (160,0 570x160)
    Rectangle (220,40 410x30), "%s", tooltip "'whitelist: Begriff1[;Begriff2[;Begriff3]]'", text variable: fbLogger.szVisuFilterWhite, colour toggle: fbLogger.bVisuFilterWhiteEnable
        OnMouseClick: execute { fbLogger.bVisuFilterWhiteEnable := TRUE; }
        OnMouseClick: write the text variable via Default
    Button (180,120 140x30), "Alle", colour toggle: fbLogger.iVisuFilterMsgTypInput <= 0
        OnMouseDown: execute { fbLogger.iVisuFilterMsgTypInput := 0; }
    Rectangle (670,40 40x30), "del", tooltip "löschen"
        OnMouseClick: execute { fbLogger.szVisuFilterWhite := ''; }
    Button (330,120 140x30), "Warnungen", colour toggle: fbLogger.iVisuFilterMsgTypInput = 1
        OnMouseDown: execute { fbLogger.iVisuFilterMsgTypInput := 1; }
    Button (480,120 140x30), "Fehlermeldungen", colour toggle: fbLogger.iVisuFilterMsgTypInput = 2
        OnMouseDown: execute { fbLogger.iVisuFilterMsgTypInput := 2; }
    Rectangle (220,80 410x30), "%s", tooltip "'black list: Begriff1[;Begriff2[;Begriff3]]'", text variable: fbLogger.szVisuFilterBlack, colour toggle: fbLogger.bVisuFilterBlackEnable
        OnMouseClick: execute { fbLogger.bVisuFilterBlackEnable := TRUE; }
        OnMouseClick: write the text variable via Default
    Rectangle (670,80 40x30), "del", tooltip "löschen"
        OnMouseClick: execute { fbLogger.szVisuFilterBlack := ''; }
    Rectangle (630,40 40x30), "...", tooltip "speichern/laden"
        OnMouseClick: execute { fbLogger.bVisuFilterWhiteEnable := TRUE; }
        OnMouseClick: change screen: V_LoggerFilterWhite
    Rectangle (630,80 40x30), "...", tooltip "speichern/laden"
        OnMouseClick: execute { fbLogger.bVisuFilterBlackEnable := TRUE; }
        OnMouseClick: change screen: V_LoggerFilterBlack
    Rectangle (0,0 160x160)
    Button (10,80 60x40), "<", invisible if: fbLogger.bVisuPrevPageInVisible
        toggle fbLogger.bVisuPrevPage
    Button (80,80 60x40), ">", invisible if: fbLogger.bVisuNextPageInVisible
        toggle fbLogger.bVisuNextPage
    Button (10,30 130x40), "Start", colour toggle: fbLogger.bVisuStart
        toggle fbLogger.bVisuStart
    Rectangle (0,160 50x40), "Id"
    Rectangle (50,160 680x40), "Message (Datum, Uhrzeit, Pfad, Text)"
    Frame (0,200 730x20)
        shows V_LoggerMsgLine(IOstLogMsg := fbLogger.astVisuLogMsg[1], IOiLogIdAct := fbLogger.nviLogId)
    Frame (0,220 730x20)
        shows V_LoggerMsgLine(IOstLogMsg := fbLogger.astVisuLogMsg[2], IOiLogIdAct := fbLogger.nviLogId)
    Frame (0,240 730x20)
        shows V_LoggerMsgLine(IOstLogMsg := fbLogger.astVisuLogMsg[3], IOiLogIdAct := fbLogger.nviLogId)
    Frame (0,260 730x20)
        shows V_LoggerMsgLine(IOstLogMsg := fbLogger.astVisuLogMsg[4], IOiLogIdAct := fbLogger.nviLogId)
    Frame (0,280 730x20)
        shows V_LoggerMsgLine(IOstLogMsg := fbLogger.astVisuLogMsg[5], IOiLogIdAct := fbLogger.nviLogId)
    Frame (0,300 730x20)
        shows V_LoggerMsgLine(IOstLogMsg := fbLogger.astVisuLogMsg[6], IOiLogIdAct := fbLogger.nviLogId)
    Frame (0,320 730x20)
        shows V_LoggerMsgLine(IOstLogMsg := fbLogger.astVisuLogMsg[7], IOiLogIdAct := fbLogger.nviLogId)
    Frame (0,340 730x20)
        shows V_LoggerMsgLine(IOstLogMsg := fbLogger.astVisuLogMsg[8], IOiLogIdAct := fbLogger.nviLogId)
    Frame (0,360 730x20)
        shows V_LoggerMsgLine(IOstLogMsg := fbLogger.astVisuLogMsg[9], IOiLogIdAct := fbLogger.nviLogId)
    Frame (0,380 730x20)
        shows V_LoggerMsgLine(IOstLogMsg := fbLogger.astVisuLogMsg[10], IOiLogIdAct := fbLogger.nviLogId)
    Rectangle (500,160 230x20), "Letzter Logeintrag: %s", text variable: fbLogger.nviLogId
    Rectangle (500,180 230x20), "Auswertung gestartet ab Logeintrag: %s", text variable: fbLogger.iVisuLogIdStart
    Rectangle (160,0 120x30), "Filter:"
    Button (420,160 70x40), "Error", invisible if: fbLogger.bVisuError = 0
    Frame (0,400 730x20)
        shows V_LoggerMsgLine(IOstLogMsg := fbLogger.astVisuLogMsg[11], IOiLogIdAct := fbLogger.nviLogId)
    Line (50,420) (50,200)
    Rectangle (180,40 40x30), "white", colour toggle: fbLogger.bVisuFilterWhiteEnable
        OnMouseClick: execute { fbLogger.bVisuFilterWhiteEnable := NOT fbLogger.bVisuFilterWhiteEnable; fbLogger.bVisuStart := TRUE; }
    Rectangle (670,10 40x30), "/", colour toggle: fbLogger.bVisuFilterWhiteMode_OR
        OnMouseClick: execute {
            fbLogger.bVisuFilterWhiteMode_OR := TRUE;
            fbLogger.bVisuFilterWhiteEnable := TRUE;
            fbLogger.bVisuStart := TRUE;
        }
    Rectangle (630,10 40x30), "&", colour toggle: fbLogger.bVisuFilterWhiteMode_OR
        OnMouseClick: execute {
            fbLogger.bVisuFilterWhiteMode_OR := FALSE;
            fbLogger.bVisuFilterWhiteEnable := TRUE;
            fbLogger.bVisuStart := TRUE;
        }
    Rectangle (180,80 40x30), "black", colour toggle: fbLogger.bVisuFilterBlackEnable
        OnMouseClick: execute { fbLogger.bVisuFilterBlackEnable := NOT fbLogger.bVisuFilterBlackEnable; fbLogger.bVisuStart := TRUE; }
    Rectangle (0,420 730x90)
    Rectangle (10,430 390x30), "Log-Datei: %s_ n.csv", text variable: fbLogger.fbFileWriteLogString.INszFileName, colour toggle: fbLogger.OUTbFileOpen
    Button (500,470 210x30), "Datenspeicherung aktivieren", tooltip "Daten werden automatisch gespeichert, wenn eine Mindestanzahl ungespeicherter Meldungen vorhanden ist.", colour toggle: fbLogger.nvbVisuFileWritingEnable
        toggle fbLogger.nvbVisuFileWritingEnable
    Button (330,470 160x30), "Daten speichern", tooltip "Daten sofort speichern", colour toggle: fbLogger.bVisuWriteToFileStart, invisible if: fbLogger.nvbVisuFileWritingEnable = 0
        OnMouseClick: execute { fbLogger.bVisuWriteToFileStart := TRUE; }
    Rectangle (10,460 230x20), "Letzter Logeintrag in Datei: %s", text variable: fbLogger.nviLogIdFileWriter
    Rectangle (10,480 220x20), "Nicht gespeicherte Logeinträge: %s", text variable: fbLogger.iFileWriterNumOfMsgsOpen, invisible if: fbLogger.nvbVisuFileWritingEnable = 0
    Button (500,430 210x30), "Speichern auf Netzwerkpfad", tooltip "Daten werden automatisch gespeichert, wenn eine Mindestanzahl ungespeicherter Meldungen vorhanden ist.", colour toggle: fbLogger.bVisuInitPathNetwork
        toggle fbLogger.bVisuInitPathNetwork
END_VISUALIZATION

// ---- Logger/VISUs/V_LoggerMsgLine.TcVIS
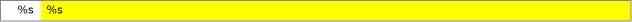
VISUALIZATION V_LoggerMsgLine  // 632x22
VAR_IN_OUT
	IOstLogMsg : ST_LogMessageVisu;
	IOiLogIdAct : INT;
END_VAR
    Rectangle (0,0 40x20)
    Rectangle (30,0 600x20)
    Rectangle (40,0 590x20), colour toggle: IOstLogMsg.iTyp > 1, invisible if: IOstLogMsg.iTyp < 1
    Rectangle (0,0 40x20), "%s", text variable: IOstLogMsg.iLogId, colour toggle: IOstLogMsg.iLogId = IOiLogIdAct, invisible if: IOstLogMsg.iLogId = 0
    Rectangle (40,0 590x20), "%s", text variable: IOstLogMsg.szLogMsg
END_VISUALIZATION

// ---- Visualizations/Frames/V_Dialog_Mob.TcVIS
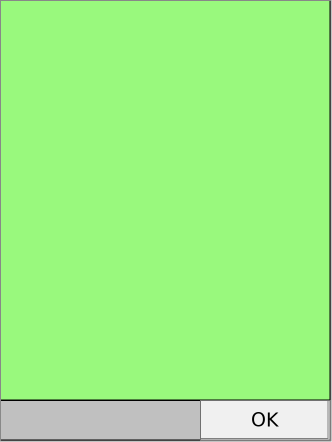
VISUALIZATION V_Dialog_Mob  // 332x442
    Rectangle (0,400 330x40)
    Rectangle (0,0 330x400)
    Button (200,400 130x40), "OK"
        OnMouseUp: change screen: Previous 
END_VISUALIZATION

// ---- Visualizations/Frames/V_Main_Mob.TcVIS
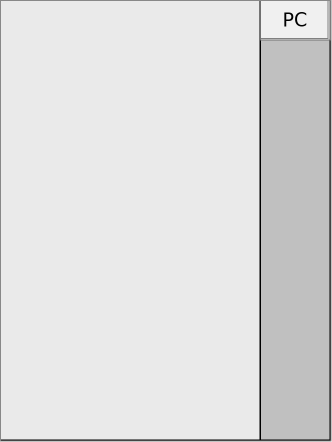
VISUALIZATION V_Main_Mob  // 332x442
    Rectangle (260,0 70x440)
    Rectangle (0,0 260x440)
    Button (260,0 70x40), "PC"
        OnMouseUp: change screen: V_Main_PC
END_VISUALIZATION

// ---- Visualizations/Frames/V_Main_PC.TcVIS
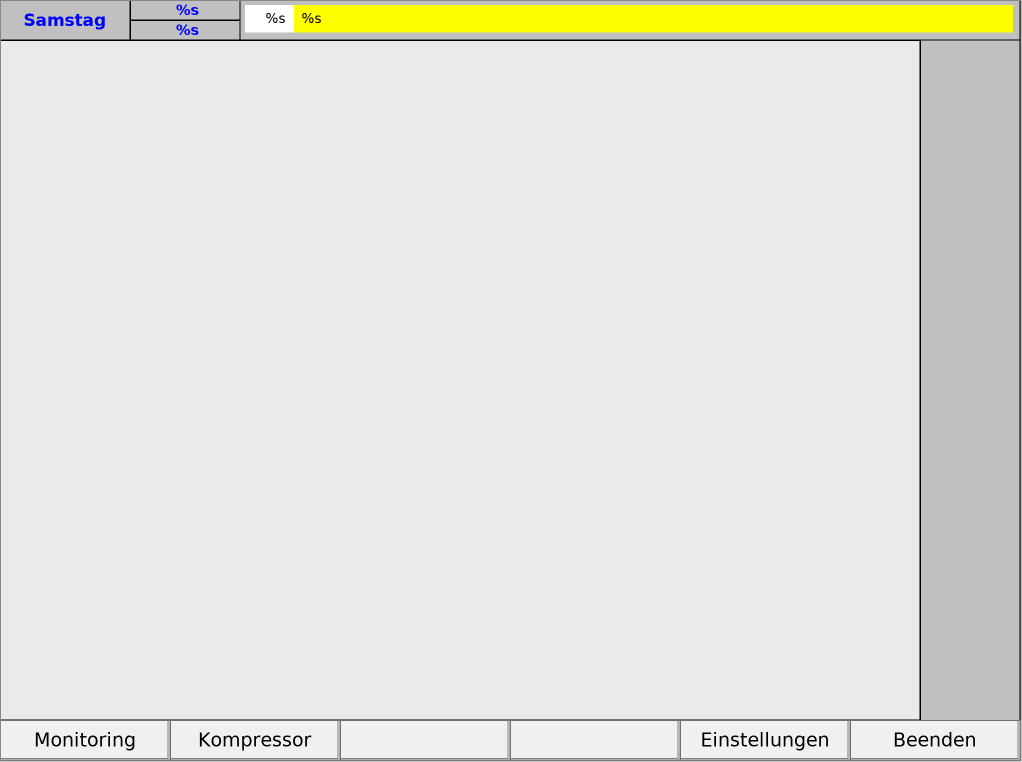
VISUALIZATION V_Main_PC  // 1022x762
    Rectangle (920,30 100x730)
    Rectangle (0,0 1020x40)
    Rectangle (0,40 920x680)
    Rectangle (0,720 1020x40)
    Rectangle (130,0 110x20), "%s", text variable: gfbSystemCX.OUTszDate
    Rectangle (130,20 110x20), "%s", text variable: gfbSystemCX.OUTszClock
    Button (850,720 170x40), "Beenden"
    Button (680,720 170x40), "Einstellungen"
        OnMouseUp: change screen: V_Einstellungen
    Button (510,720 170x40)
    Button (340,720 170x40)
    Button (0,720 170x40), "Monitoring"
        OnMouseUp: change screen: V_Monitoring
    Rectangle (0,0 130x40), "Sonntag", invisible if: gfbSystemCX.OUTeDayOfWeek > 0
    Rectangle (0,0 130x40), "Montag", invisible if: gfbSystemCX.OUTeDayOfWeek <> 1
    Rectangle (0,0 130x40), "Dienstag", invisible if: gfbSystemCX.OUTeDayOfWeek <> 2
    Rectangle (0,0 130x40), "Mittwoch", invisible if: gfbSystemCX.OUTeDayOfWeek <> 3
    Rectangle (0,0 130x40), "Donnerstag", invisible if: gfbSystemCX.OUTeDayOfWeek <> 4
    Rectangle (0,0 130x40), "Freitag", invisible if: gfbSystemCX.OUTeDayOfWeek <> 5
    Rectangle (0,0 130x40), "Samstag", invisible if: gfbSystemCX.OUTeDayOfWeek <> 6
    Frame (245,5 770x30)
        shows V_LoggerMsgLine(IOstLogMsg := gfbLogger.nvstVisuActualMessage, IOiLogIdAct := gfbLogger.nviLogId)
        OnMouseClick: change screen: V_Logger
        OnMouseDown: execute { gfbLogger.bVisuStart := TRUE; }
    Button (170,720 170x40), "Kompressor"
        OnMouseUp: change screen: V_KomprWRG
END_VISUALIZATION

// ---- Visualizations/Module/V_ECReset.TcVIS
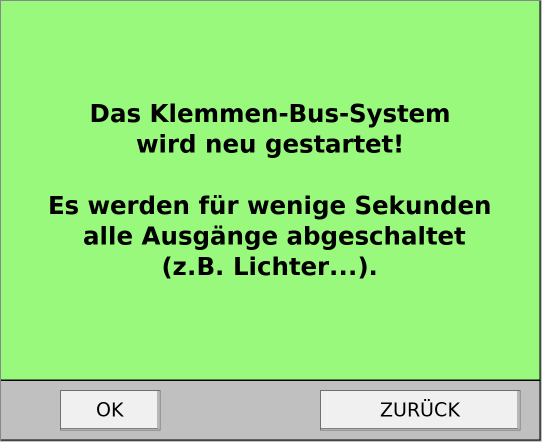
VISUALIZATION V_ECReset  // 542x442
    Rectangle (0,380 540x60)
    Button (60,390 100x40), "OK"
        OnMouseDown: toggle gfbSystemCX.VbDeviceReset
        OnMouseUp: change screen: Previous 
    Button (320,390 200x40), "ZURÜCK"
        OnMouseUp: change screen: Previous 
    Rectangle (0,0 540x380), "Das Klemmen-Bus-System wird neu gestartet! Es werden für wenige Sekunden alle Ausgänge abgeschaltet (z.B. Lichter...)."
END_VISUALIZATION

// ---- Visualizations/Module/V_LiquidSensorCfg.TcVIS
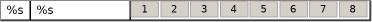
VISUALIZATION V_LiquidSensorCfg  // 372x22
VAR_INPUT
  iNumOfCh : INT;
END_VAR
VAR_IN_OUT
	IOfbLiquidSensor : FB_LiquidSensor;
END_VAR
    Rectangle (130,0 240x20)
    Rectangle (0,0 30x20), "%s", text variable: IOfbLiquidSensor.iChan
    Rectangle (30,0 100x20), "%s", text variable: IOfbLiquidSensor.VnvszName
        OnMouseDown: write the text variable via Default
    Frame (130,0 239x19)
        shows V_dwBitToggle(iNumOfCh := iNumOfCh, dwVar := IOfbLiquidSensor.VnvdwCFGLiquidToTransor)
END_VISUALIZATION

// ---- Visualizations/Module/V_LiquidSensorState.TcVIS
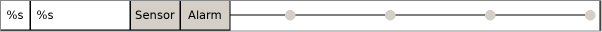
VISUALIZATION V_LiquidSensorState  // 602x32
VAR_IN_OUT
	IOfbLiquidSensor : FB_LiquidSensor;
END_VAR
    Line (590,15) (230,15), colour toggle: IOfbLiquidSensor.QbLMStatus, invisible if: IOfbLiquidSensor.VnvdwCFGLiquidToTransor.4 = 0
    Ellipse (585,10 10x10), colour toggle: IOfbLiquidSensor.QbLMStatus, invisible if: IOfbLiquidSensor.VnvdwCFGLiquidToTransor.4 = 0
    Line (490,15) (230,15), colour toggle: IOfbLiquidSensor.QbLMStatus, invisible if: IOfbLiquidSensor.VnvdwCFGLiquidToTransor.3 = 0
    Ellipse (485,10 10x10), colour toggle: IOfbLiquidSensor.QbLMStatus, invisible if: IOfbLiquidSensor.VnvdwCFGLiquidToTransor.3 = 0
    Line (390,15) (230,15), colour toggle: IOfbLiquidSensor.QbLMStatus, invisible if: IOfbLiquidSensor.VnvdwCFGLiquidToTransor.2 = 0
    Ellipse (385,10 10x10), colour toggle: IOfbLiquidSensor.QbLMStatus, invisible if: IOfbLiquidSensor.VnvdwCFGLiquidToTransor.2 = 0
    Rectangle (0,0 30x30), "%s", text variable: IOfbLiquidSensor.iChan
    Rectangle (30,0 100x30), "%s", text variable: IOfbLiquidSensor.VnvszName
    Rectangle (180,0 50x30), "Alarm", colour toggle: IOfbLiquidSensor.QbLMStatus
    Line (290,15) (230,15), colour toggle: IOfbLiquidSensor.QbLMStatus, invisible if: IOfbLiquidSensor.VnvdwCFGLiquidToTransor.1 = 0
    Ellipse (285,10 10x10), colour toggle: IOfbLiquidSensor.QbLMStatus, invisible if: IOfbLiquidSensor.VnvdwCFGLiquidToTransor.1 = 0
    Line (600,30) (600,0)
    Rectangle (130,0 50x30), "Sensor", colour toggle: IOfbLiquidSensor.IbLiquidSensor
END_VISUALIZATION

// ---- Visualizations/Module/V_LiquidTransorState.TcVIS
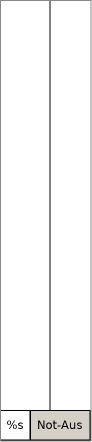
VISUALIZATION V_LiquidTransorState  // 92x442
VAR_IN_OUT
	IOfbTransor : FB_Transor;
END_VAR
    Rectangle (0,410 30x30), "%s", text variable: IOfbTransor.iChan
    Rectangle (30,410 60x30), "Not-Aus", colour toggle: IOfbTransor.QbTransor
    Line (50,410) (50,0), colour toggle: IOfbTransor.QbTransor
END_VISUALIZATION

// ---- Visualizations/Module/V_NumInputReal.TcVIS
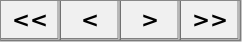
VISUALIZATION V_NumInputReal  // 242x42
VAR_INPUT
	INrValueMin		: REAL;
	INrValueMax		: REAL;
	INrStepMin		: REAL;
	INrStepMax		: REAL;
END_VAR
VAR_IN_OUT
	INrVariable		: REAL;
END_VAR
    Button (120,0 60x40), ">", invisible if: INrVariable >= INrValueMax
        OnMouseClick: execute {
            INrVariable :=
            	INrVariable
            	+ INrStepMin;
        }
    Button (60,0 60x40), "<", invisible if: INrVariable <= INrValueMin
        OnMouseClick: execute {
            INrVariable :=
            	INrVariable
            	- INrStepMin;
        }
    Button (180,0 60x40), ">>", invisible if: INrVariable >= INrValueMax
        OnMouseClick: execute {
            INrVariable :=
            	INrVariable
            	+ INrStepMax;
        }
    Button (0,0 60x40), "<<", invisible if: INrVariable <= INrValueMin
        OnMouseClick: execute {
            INrVariable :=
            	INrVariable
            	- INrStepMax;
        }
END_VISUALIZATION

// ---- Visualizations/Module/V_RadioButton.TcVIS
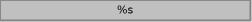
VISUALIZATION V_RadioButton  // 252x22
VAR_INPUT
	IN_Title		: STRING;
	IN_iValue		: INT;
END_VAR
VAR_IN_OUT
	IO_iVar 		: INT;
END_VAR
    Rectangle (0,0 250x20), "%s", text variable: IN_Title, colour toggle: IO_iVar = IN_iValue
        OnMouseClick: execute { IO_iVar := IN_iValue; }
END_VISUALIZATION

// ---- Visualizations/Module/V_TCReset.TcVIS
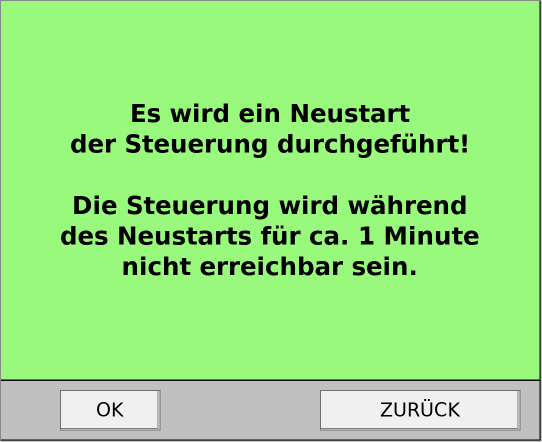
VISUALIZATION V_TCReset  // 542x442
vAR_IN_OUT
	
END_VAR
    Rectangle (0,380 540x60)
    Button (60,390 100x40), "OK"
        OnMouseUp: change screen: Previous 
        OnMouseDown: toggle gfbSystemCX.VbTCReset
    Button (320,390 200x40), "ZURÜCK"
        OnMouseUp: change screen: Previous 
    Rectangle (0,0 540x380), "Es wird ein Neustart der Steuerung durchgeführt! Die Steuerung wird während des Neustarts für ca. 1 Minute nicht erreichbar sein."
END_VISUALIZATION

// ---- Visualizations/Module/V_WCRaum.TcVIS
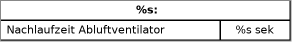
VISUALIZATION V_WCRaum  // 292x42
VAR_INPUT
	IN_Title		: STRING;
END_VAR
VAR_IN_OUT
	IO_fbWCRaum : FB_WCRaum;
END_VAR
    Rectangle (220,20 70x20), "%s sek", tooltip "Nach Abschalten des Bewegungsmelders läuft der Abluftventilator die hier eingestellte Zeit nach", text variable: IO_fbWCRaum.VdiAbluftNachlaufzeit
        OnMouseClick: write the text variable via Default, min 3, max 2000
    Rectangle (0,20 220x20), "Nachlaufzeit Abluftventilator", tooltip "Nach Abschalten des Bewegungsmelders läuft der Abluftventilator die hier eingestellte Zeit nach"
    Rectangle (0,0 290x20), "%s:", tooltip "Nach Abschalten des Bewegungsmelders läuft der Abluftventilator die hier eingestellte Zeit nach", text variable: IN_Title
END_VISUALIZATION

// ---- Visualizations/Module/V_WeekDay.TcVIS
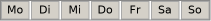
VISUALIZATION V_WeekDay  // 211x21
VAR_IN_OUT
	eWeekDay : E_WeekDay;
END_VAR
    Rectangle (1,1 28x18), "Mo", colour toggle: eWeekDay = 1
        OnMouseUp: execute { eWeekDay := 1; }
    Rectangle (31,1 28x18), "Di", colour toggle: eWeekDay = 2
        OnMouseUp: execute { eWeekDay := 2; }
    Rectangle (61,1 28x18), "Mi", colour toggle: eWeekDay = 3
        OnMouseUp: execute { eWeekDay := 3; }
    Rectangle (91,1 28x18), "Do", colour toggle: eWeekDay = 4
        OnMouseUp: execute { eWeekDay := 4; }
    Rectangle (121,1 28x18), "Fr", colour toggle: eWeekDay = 5
        OnMouseUp: execute { eWeekDay := 5; }
    Rectangle (151,1 28x18), "Sa", colour toggle: eWeekDay = 6
        OnMouseUp: execute { eWeekDay := 6; }
    Rectangle (181,1 28x18), "So", colour toggle: eWeekDay = 0
        OnMouseUp: execute { eWeekDay := 0; }
END_VISUALIZATION

// ---- Visualizations/Module/V_dwBitToggle.TcVIS
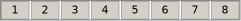
VISUALIZATION V_dwBitToggle  // 241x21
VAR_INPUT
  iNumOfCh : INT;
END_VAR
VAR_IN_OUT
	dwVar : DWORD;
END_VAR
    Rectangle (1,1 28x18), "1", colour toggle: dwVar.1, invisible if: iNumOfCh < 1
        toggle dwVar.1
    Rectangle (31,1 28x18), "2", colour toggle: dwVar.2, invisible if: iNumOfCh < 2
        toggle dwVar.2
    Rectangle (61,1 28x18), "3", colour toggle: dwVar.3, invisible if: iNumOfCh < 3
        toggle dwVar.3
    Rectangle (91,1 28x18), "4", colour toggle: dwVar.4, invisible if: iNumOfCh < 4
        toggle dwVar.4
    Rectangle (121,1 28x18), "5", colour toggle: dwVar.5, invisible if: iNumOfCh < 5
        toggle dwVar.5
    Rectangle (151,1 28x18), "6", colour toggle: dwVar.6, invisible if: iNumOfCh < 6
        toggle dwVar.6
    Rectangle (181,1 28x18), "7", colour toggle: dwVar.7, invisible if: iNumOfCh < 7
        toggle dwVar.7
    Rectangle (211,1 28x18), "8", colour toggle: dwVar.8, invisible if: iNumOfCh < 8
        toggle dwVar.8
END_VISUALIZATION

// ---- Visualizations/VisuStart.TcVIS
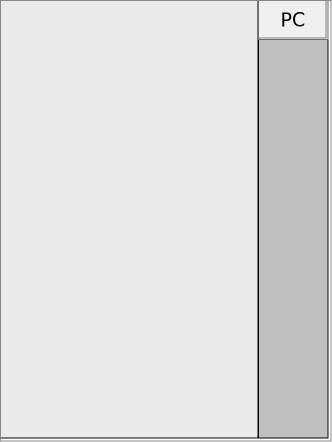
VISUALIZATION VisuStart  // 332x442
    Frame (0,0 330x440)
        shows V_Main_Mob()
END_VISUALIZATION

// ---- Visualizations/Module/V_Heizung.TcVIS
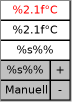
VISUALIZATION V_Heizung  // 72x102
VAR_IN_OUT
	m_Input_fbHeizregler : FB_Heizregler;
END_VAR
    Rectangle (0,60 50x20), "%s%%", text variable: m_Input_fbHeizregler.iManPHeiz, colour toggle: (m_Input_fbHeizregler.bManuell) <> 0
        OnMouseDown: write the text variable via Default
    Rectangle (0,80 50x20), "Manuell", colour toggle: (m_Input_fbHeizregler.bManuell) <> 0
        toggle m_Input_fbHeizregler.bManuell
    Rectangle (0,0 70x20), "%2.1f°C", text variable: m_Input_fbHeizregler.diTempIst * 0.01
    Rectangle (0,20 70x20), "%2.1f°C", text variable: m_Input_fbHeizregler.diTempSoll * 0.01
    Rectangle (0,40 70x20), "%s%%", text variable: m_Input_fbHeizregler.iPHeiz
        OnMouseDown: write the text variable via Edit
    Rectangle (50,60 20x20), "+", colour toggle: (m_Input_fbHeizregler.bManuell) <> 0
        OnMouseClick: execute {
            IF (m_Input_fbHeizregler.iManPHeiz < 95) THEN
            	m_Input_fbHeizregler.iManPHeiz :=
            		m_Input_fbHeizregler.iManPHeiz
            		+ 5;
            ELSE
            	m_Input_fbHeizregler.iManPHeiz := 100;
            END_IF
        }
    Rectangle (50,80 20x20), "-", colour toggle: (m_Input_fbHeizregler.bManuell) <> 0
        OnMouseClick: execute {
            IF (m_Input_fbHeizregler.iManPHeiz > 5) THEN
            	m_Input_fbHeizregler.iManPHeiz :=
            		m_Input_fbHeizregler.iManPHeiz
            		- 5;
            ELSE
            	m_Input_fbHeizregler.iManPHeiz := 0;
            END_IF
        }
END_VISUALIZATION

// ---- Visualizations/Module/V_Licht.TcVIS
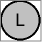
VISUALIZATION V_Licht  // 42x42
VAR_IN_OUT
	m_Input_fbLicht : FB_Licht;
END_VAR
    Ellipse (0,0 40x40), "L", colour toggle: (m_Input_fbLicht.QbOutLicht) <> 0
        tap m_Input_fbLicht.bInVisu
    Polyline (30,30)
    Polyline (0,0)
    Polyline (30,10)
    Polyline (10,30)
END_VISUALIZATION

// ---- Visualizations/Module/V_Rol.TcVIS
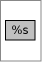
VISUALIZATION V_Rol  // 42x62
VAR_IN_OUT
	m_Input_fbRollo : FB_Rollo;
END_VAR
    Polygon (0,20)
    Polygon (0,20), invisible if: (m_Input_fbRollo.bOutRollo =0) <> 0
    Polygon (40,20), invisible if: (m_Input_fbRollo.bOutVisuAb =0) <> 0
    Polygon (40,40), invisible if: (m_Input_fbRollo.bOutVisuAb =1) <> 0
    Rectangle (5,20 30x20), "%s", text variable: m_Input_fbRollo.iActPos, colour toggle: (m_Input_fbRollo.bOutRollo) <> 0
    Polygon (40,20), colour toggle: (m_Input_fbRollo.bInVisuAuf) <> 0
        tap m_Input_fbRollo.bInVisuAuf
    Polygon (20,60), colour toggle: (m_Input_fbRollo.bInVisuAb) <> 0
        tap m_Input_fbRollo.bInVisuAb
END_VISUALIZATION

// ---- Visualizations/Module/V_RolGrp.TcVIS
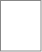
VISUALIZATION V_RolGrp  // 42x52
VAR_IN_OUT
	m_Input_fbRolloGruppe : FB_RolloGruppe;
END_VAR
    Polygon (40,20), colour toggle: (m_Input_fbRolloGruppe.tonRolloAb.Q =0) <> 0, invisible if: (m_Input_fbRolloGruppe.QbOutRolloAb =1) <> 0
    Polygon (40,30), colour toggle: (m_Input_fbRolloGruppe.tonRolloAb.Q =0) <> 0, invisible if: (m_Input_fbRolloGruppe.QbOutRolloAb =0) <> 0
    Polygon (40,20), colour toggle: (m_Input_fbRolloGruppe.bInVisuAuf) <> 0
        tap m_Input_fbRolloGruppe.bInVisuAuf
    Polygon (20,50), colour toggle: (m_Input_fbRolloGruppe.bInVisuAb) <> 0
        tap m_Input_fbRolloGruppe.bInVisuAb
END_VISUALIZATION

// ---- Visualizations/V_Monitoring.TcVIS
